// TwinCAT 3 PLC project SampleSymbols
// ProgramVersion: 3.1.4023.0
// libraries:
//   Tc2_Standard, * (Beckhoff Automation GmbH)
//   Tc2_System, * (Beckhoff Automation GmbH)
//   Tc3_Module, * (Beckhoff Automation GmbH)
// project tree:
//   DUTs/ LoremItem.TcDUT (not stored), LoremProperties.TcDUT
//   / PlcTask.TcTTO (not stored)
//   POUs/ MAIN.TcPOU (not stored)

// ---- DUTs/LoremProperties.TcDUT
TYPE LoremProperties :
STRUCT
	length: INT;
	hasUppercase: BOOL;
	chars: ARRAY [0..255] OF STRING;
END_STRUCT
END_TYPE
